TYPE DUT_GetBitting :
STRUCT
	CodeSchema				: STRING(50);
	SideBar					: STRING(50);
END_STRUCT
END_TYPE

(* stored: Version 1.1.0.1, ProductVersion 3.1.4024.15
   DUT DUT_GetBitting: Id {75c16cc5-f363-4afa-b131-e61e70b99b83} *)
